(* Schneider Machine Expert - Basic project s, file version 2.0.0.0 *)
(* ProjectInformations: Name=New project *)

HARDWARE
  Cpu 0: TM221CE16R
  EthernetConfiguration: NetworkName=M221, IpAllocationMode=FixedAddress, IpAddress=0.0.0.0, SubnetMask=0.0.0.0
  SerialLineConfiguration: Baud=Baud19200, Parity=ParityEven, DataBits=DataBits8, StopBits=StopBits1, PhysicalMedium=PhysicalMediumRs485, TransmissionMode=TransmissionModeModbusRtu, SlaveId=1, Addressing=SlaveAddressing
  MastTask: UsePeriodScanMode=false, PeriodScan=100
  FastTask: Period=255
  CpuBehavior: StartingMode=StartAsPreviousState, AutoSaveRamOnEeprom=true, WatchdogPeriod=250

SYMBOLS  (address, symbol, comment, settings)
  %S0       SB_COLDSTART  "Indicates or executes a cold start (data initialized to default values)"
  %S1       SB_WARMSTART  "Indicates there was a warm start with data backup"
  %S4       SB_TB10MS  "Time base of 10 ms generated by an internal clock"
  %S5       SB_TB100MS  "Time base of 100 ms generated by an internal clock"
  %S6       SB_TB1S  "Time base of 1 s generated by an internal clock"
  %S7       SB_TB1MIN  "Time base of 1 min generated by an internal clock"
  %S17      SB_LASTBIT  "It indicates the value of the last ejected bit"
  %S18      SB_OPERROR  "It indicates an overflow when a 16 bit operation is performed"
  %S19      SB_OVERRUN  "It indicates scan time greater than the period defined by the user"
  %S20      SB_INDERROR  "This bit indicates an index overflow of the indexed object address when a 16 bit operation is performed"

POU New POU
  (* SectionNumber=1 *)

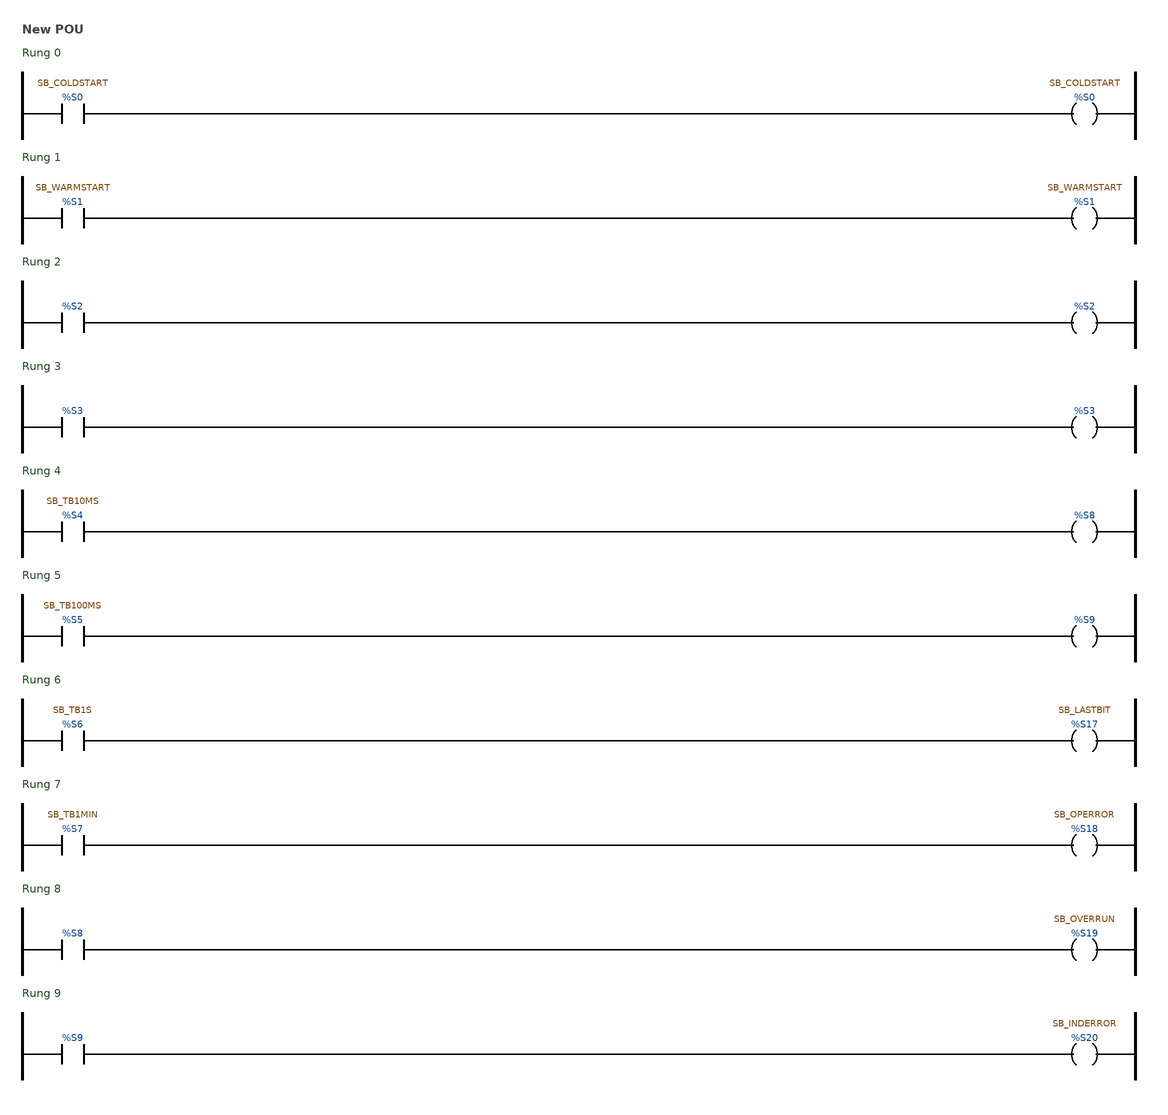

// Rung 0
  LD %S0                  (* SB_COLDSTART *)
  ST %S0                  (* SB_COLDSTART *)
  // as ST:
  //   SB_COLDSTART := SB_COLDSTART;

// Rung 1
  LD %S1                  (* SB_WARMSTART *)
  ST %S1                  (* SB_WARMSTART *)
  // as ST:
  //   SB_WARMSTART := SB_WARMSTART;

// Rung 2
  LD %S2
  ST %S2
  // as ST:
  //   %S2 := %S2;

// Rung 3
  LD %S3
  ST %S3
  // as ST:
  //   %S3 := %S3;

// Rung 4
  LD %S4                  (* SB_TB10MS *)
  ST %S8
  // as ST:
  //   %S8 := SB_TB10MS;

// Rung 5
  LD %S5                  (* SB_TB100MS *)
  ST %S9
  // as ST:
  //   %S9 := SB_TB100MS;

// Rung 6
  LD %S6                  (* SB_TB1S *)
  ST %S17                 (* SB_LASTBIT *)
  // as ST:
  //   SB_LASTBIT := SB_TB1S;

// Rung 7
  LD %S7                  (* SB_TB1MIN *)
  ST %S18                 (* SB_OPERROR *)
  // as ST:
  //   SB_OPERROR := SB_TB1MIN;

// Rung 8
  LD %S8
  ST %S19                 (* SB_OVERRUN *)
  // as ST:
  //   SB_OVERRUN := %S8;

// Rung 9
  LD %S9
  ST %S20                 (* SB_INDERROR *)
  // as ST:
  //   SB_INDERROR := %S9;
